ABB RobotStudio station: PROYECTO FINAL_TERMINADO_1.rsstn

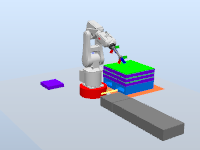
Station PROYECTO FINAL_TERMINADO (saved by RobotStudio 20.1.9014.1)
Controller Controller1, task T_ROB1: task frame (RAPID world) sits at (0, 0, 100) mm in the station
Controller Controller1
  mechanical unit ROB_1: IRB120_3_58__01, 6 joints, base frame (0, 0, 0) mm
Layout (positions relative to the parent item):
  - IRB120_3_58__01 [mechanism, from Robots\IRB120_3_58_G_01.rslib] at (0, 0, 100) mm; joint values [0, -0.0243, 0.3487, 0, 0.1992, 0] (rad or m)
  - soporte [mechanism, from biblioteca de robot\soporte.rslib] at (364.35, 0, 594) mm, rotated rx 180 ry 60 rz 180 deg
  - caja_modelo [part] at (-385.91, -352.84, 0) mm, rotated rx 0 ry 0 rz -0.36 deg
  - tapa_nueva3 [part] at (247.21, 259.23, 238) mm
  - pale_nuevo [part] at (30.71, 458.19, 106.32) mm
  - tapa_nueva2 [part] at (33.05, 460.18, 197.68) mm
  - tapa_nueva1 [part] at (31.05, 458.19, 150.3) mm
  - base_robot [part]
  - reposicion [smart component]
      signals: DI reseteo
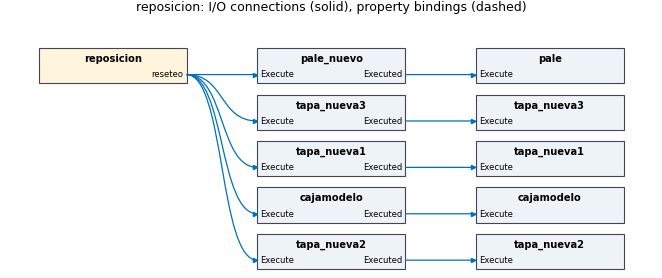
      connections:
        reposicion.reseteo -> pale_nuevo.Execute
        reposicion.reseteo -> tapa_nueva3.Execute
        reposicion.reseteo -> tapa_nueva1.Execute
        reposicion.reseteo -> cajamodelo.Execute
        reposicion.reseteo -> tapa_nueva2.Execute
        tapa_nueva2.Executed -> tapa_nueva2.Execute
        cajamodelo.Executed -> cajamodelo.Execute
        tapa_nueva1.Executed -> tapa_nueva1.Execute
        tapa_nueva3.Executed -> tapa_nueva3.Execute
        pale_nuevo.Executed -> pale.Execute
    - pale_nuevo [smart component, from Components\Positioner.rslib]
        properties: Object=pale_nuevo; Position=[0.061428 -0.45 0.13]; Orientation=[0 0 0]; Reference=Global; ReferenceObject=(none)
    - tapa_nueva1 [smart component, from Components\Positioner.rslib]
        properties: Object=tapa_nueva1; Position=[0.061428 -0.45 0.03]; Orientation=[0 0 0]; Reference=Global; ReferenceObject=(none)
    - tapa_nueva2 [smart component, from Components\Positioner.rslib]
        properties: Object=tapa_nueva2; Position=[0.061428 -0.45 0.018]; Orientation=[0 0 0]; Reference=Global; ReferenceObject=(none)
    - tapa_nueva3 [smart component, from Components\Positioner.rslib]
        properties: Object=tapa_nueva3; Position=[0.276428 -0.65 0]; Orientation=[0 0 0]; Reference=Global; ReferenceObject=(none)
    - cajamodelo [smart component, from Components\Positioner.rslib]
        properties: Object=(none); Position=[2.337542 0 0.14]; Orientation=[0 0 0]; Reference=Global; ReferenceObject=(none)
    - cajamodelo [smart component, from Components\Detacher.rslib]
        properties: Child=(none); KeepPosition=true
    - pale [smart component, from Components\Detacher.rslib]
        properties: Child=pale_nuevo; KeepPosition=true
    - tapa_nueva1 [smart component, from Components\Detacher.rslib]
        properties: Child=tapa_nueva1; KeepPosition=true
    - tapa_nueva2 [smart component, from Components\Detacher.rslib]
        properties: Child=tapa_nueva2; KeepPosition=true
    - tapa_nueva3 [smart component, from Components\Detacher.rslib]
        properties: Child=tapa_nueva3; KeepPosition=true
  - pedestal [part] at (28.42, 0, 0) mm
  - superficie [part] at (-277.21, 164.21, 2) mm
  - Pieza_3 [part]
  - tapa [part] at (246.05, 1411.93, 141.43) mm
  - cajas_y_banda [smart component]
      signals: DI caja_nuevaS, DO sensorLineal, DI attcherS, DI dettacherS, DI moverCajaS
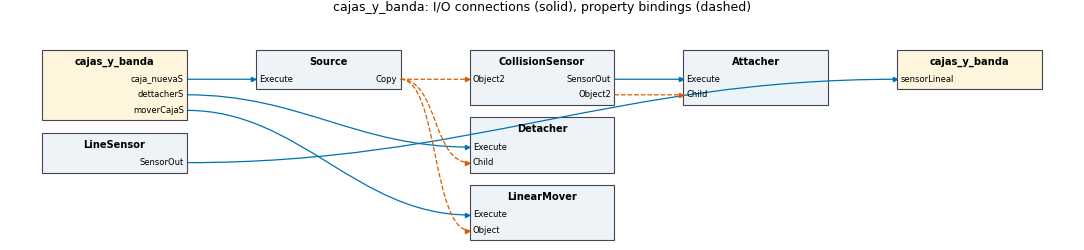
      connections:
        cajas_y_banda.caja_nuevaS -> Source.Execute
        LineSensor.SensorOut -> cajas_y_banda.sensorLineal
        cajas_y_banda.dettacherS -> Detacher.Execute
        cajas_y_banda.moverCajaS -> LinearMover.Execute
        CollisionSensor.SensorOut -> Attacher.Execute
        Source.Copy => Detacher.Child
        Source.Copy => CollisionSensor.Object2
        Source.Copy => LinearMover.Object
        CollisionSensor.Object2 => Attacher.Child
    - LineSensor [smart component, from Components\LineSensor.rslib] at (305.23, 54.67, 138.21) mm, rotated rx 90 ry 0 rz 0 deg
        properties: Start=[0.00491899596865375 -0.0182095563953858 -0.0453285878030492]; End=[0.00491899596865375 -0.0182095563953858 0.154671412196951]; Radius=0.005; SensedPart=(none); SensedPoint=[0 0 0]
      - _sensorPart_ [part]
    - LinearMover [smart component, from Components\LinearMover.rslib]
        properties: Object=caja_modelo_143; Direction=[-0.5 0 0]; Speed=0.3; Reference=Global; ReferenceObject=(none)
    - Source [smart component, from Components\Source.rslib]
        properties: Source=caja_modelo; Copy=caja_modelo_143; Parent=(none); Position=[1.18454 -0.1 0.1]; Orientation=[0 0 0]; Transient=false; PhysicsBehavior=0
    - CollisionSensor [smart component, from Components\CollisionSensor.rslib]
        properties: Object1=soporte; Object2=caja_modelo_143; NearMiss=0.002; Part1=(none); Part2=(none); CollisionType=0
    - Attacher [smart component, from Components\Attacher.rslib]
        properties: Parent=soporte; Flange=0; Child=caja_modelo_143; Mount=false; Offset=[0 0 0]; Orientation=[0 0 0]
    - Detacher [smart component, from Components\Detacher.rslib]
        properties: Child=caja_modelo_143; KeepPosition=true
  - pallet [smart component]
      connections:
        CollisionSensor.SensorOut -> Attacher.Execute
        CollisionSensor_2.SensorOut -> Detacher.Execute
    - Attacher [smart component, from Components\Attacher.rslib]
        properties: Parent=soporte; Flange=0; Child=pale_nuevo; Mount=false; Offset=[0 0 0]; Orientation=[0 0 0]
    - Detacher [smart component, from Components\Detacher.rslib]
        properties: Child=pale_nuevo; KeepPosition=true
    - CollisionSensor [smart component, from Components\CollisionSensor.rslib]
        properties: Object1=soporte; Object2=pale_nuevo; NearMiss=0.003; Part1=(none); Part2=(none); CollisionType=0
    - CollisionSensor_2 [smart component, from Components\CollisionSensor.rslib]
        properties: Object1=pale_nuevo; Object2=superficie; NearMiss=0.005; Part1=pale_nuevo; Part2=superficie; CollisionType=1
  - tapasDeNivel [smart component]
      signals: DI soltarTapa
      connections:
        CollisionSensor_3.SensorOut -> Attacher_2.Execute
        tapasDeNivel.soltarTapa -> Detacher_2.Execute
        CollisionSensor_4.SensorOut -> Attacher_3.Execute
        tapasDeNivel.soltarTapa -> Detacher_3.Execute
        CollisionSensor_5.SensorOut -> Attacher_4.Execute
        tapasDeNivel.soltarTapa -> Detacher_4.Execute
        CollisionSensor_3.Object2 => Attacher_2.Child
    - CollisionSensor_3 [smart component, from Components\CollisionSensor.rslib]
        properties: Object1=soporte; Object2=tapa_nueva1; NearMiss=0.001; Part1=(none); Part2=(none); CollisionType=0
    - Attacher_2 [smart component, from Components\Attacher.rslib]
        properties: Parent=soporte; Flange=0; Child=tapa_nueva1; Mount=false; Offset=[0 0 0]; Orientation=[0 0 0]
    - Detacher_2 [smart component, from Components\Detacher.rslib]
        properties: Child=tapa_nueva1; KeepPosition=true
    - Attacher_3 [smart component, from Components\Attacher.rslib]
        properties: Parent=soporte; Flange=0; Child=tapa_nueva2; Mount=false; Offset=[0 0 0]; Orientation=[0 0 0]
    - Detacher_3 [smart component, from Components\Detacher.rslib]
        properties: Child=tapa_nueva2; KeepPosition=true
    - CollisionSensor_4 [smart component, from Components\CollisionSensor.rslib]
        properties: Object1=soporte; Object2=tapa_nueva2; NearMiss=0.002; Part1=(none); Part2=(none); CollisionType=0
    - CollisionSensor_5 [smart component, from Components\CollisionSensor.rslib]
        properties: Object1=soporte; Object2=tapa_nueva3; NearMiss=0.001; Part1=(none); Part2=(none); CollisionType=0
    - Attacher_4 [smart component, from Components\Attacher.rslib]
        properties: Parent=soporte; Flange=0; Child=tapa_nueva3; Mount=false; Offset=[0 0 0]; Orientation=[0 0 0]
    - Detacher_4 [smart component, from Components\Detacher.rslib]
        properties: Child=tapa_nueva3; KeepPosition=true
  - Pieza_5 [part]
  - caja_modelo_132 [part] at (26.34, 258.19, 103.21) mm
  - caja_modelo_133 [part] at (27.58, 462.18, 103.22) mm
  - caja_modelo_134 [part] at (246.58, 460.85, 104.1) mm
  - caja_modelo_135 [part] at (245.34, 256.85, 104.3) mm
  - caja_modelo_136 [part] at (26.05, 460.19, 150.63) mm
  - caja_modelo_137 [part] at (245.05, 460.19, 150.37) mm
  - caja_modelo_138 [part] at (26.05, 256.19, 150.37) mm
  - caja_modelo_139 [part] at (245.05, 256.19, 150.61) mm
  - caja_modelo_140 [part] at (28.05, 462.19, 198.99) mm
  - caja_modelo_141 [part] at (248.85, 462.19, 199.65) mm
  - caja_modelo_142 [part] at (28.05, 258.19, 199.59) mm
  - caja_modelo_143 [part] at (247.05, 258.19, 199.43) mm
Attachment: soporte is attached to IRB120_3_58__01 / Link6
Station signals: DI inicioS, DI repo
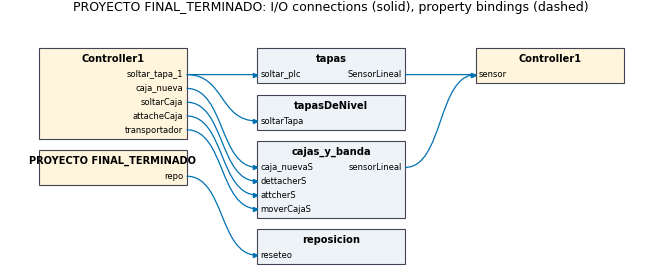
Station logic (signal -> signal, property => property):
  Controller1.soltar_tapa_1 -> tapas.soltar_plc
  anclado_y_desanclado_caja_modelo.SensorLineal -> Controller1.sensor
  cajas_y_banda.sensorLineal -> Controller1.sensor
  Controller1.caja_nueva -> cajas_y_banda.caja_nuevaS
  Controller1.soltarCaja -> cajas_y_banda.dettacherS
  Controller1.attacheCaja -> cajas_y_banda.attcherS
  Controller1.transportador -> cajas_y_banda.moverCajaS
  Controller1.soltar_tapa_1 -> tapasDeNivel.soltarTapa
  PROYECTO FINAL_TERMINADO.repo -> reposicion.reseteo
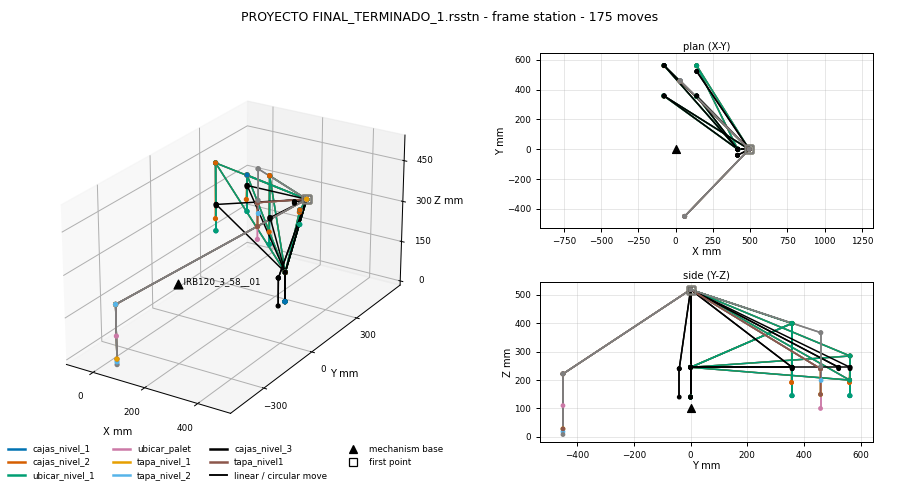
[picture p0: tool path of PROYECTO FINAL_TERMINADO_1.rsstn in frame station, 175 of 175 moves have a stored position in this frame; points joined in program order, loops and branches not executed]
Targets, tools, work objects and paths stored in the station, written as RAPID:
! task T_ROB1
MODULE CalibData
  PERS tooldata soporte:=[TRUE,[[0,0,150],[1,0,0,0]],[0.1,[0,0,1],[1,0,0,0],0,0,0]];
ENDMODULE

! task T_ROB1
MODULE Module1
  CONST robtarget pale_enposicion:=[[30.714,458.188,0],[0,1,0,0],[0,0,-2,0],[9E+09,9E+09,9E+09,9E+09,9E+09,9E+09]];
  CONST robtarget pale_enposicion_cercano:=[[30.714,458.188,140],[0,1,0,0],[0,0,-2,0],[9E+09,9E+09,9E+09,9E+09,9E+09,9E+09]];
  CONST robtarget home:=[[494.25763964,0,419],[0.5,0,0.866025404,0],[0,0,0,0],[9E+09,9E+09,9E+09,9E+09,9E+09,9E+09]];
  CONST robtarget tapa_nueva_3:=[[61.428,-450,-92],[0,1,0,0],[-1,0,1,0],[9E+09,9E+09,9E+09,9E+09,9E+09,9E+09]];
  CONST robtarget pale_nuevo:=[[61.428,-450,10],[0,1,0,0],[0,0,0,0],[9E+09,9E+09,9E+09,9E+09,9E+09,9E+09]];
  CONST robtarget tapa_nueva_1:=[[61.428,-450,-72],[0,1,0,0],[0,0,0,0],[9E+09,9E+09,9E+09,9E+09,9E+09,9E+09]];
  CONST robtarget tapa_nueva_2:=[[61.428,-450,-82],[0,1,0,0],[-1,0,1,0],[9E+09,9E+09,9E+09,9E+09,9E+09,9E+09]];
  CONST robtarget home_1:=[[417.312,0.001,268.837186077],[0,1,0,0],[0,0,-2,0],[9E+09,9E+09,9E+09,9E+09,9E+09,9E+09]];
  CONST robtarget cercano_pale_nuevo:=[[61.428,-450,121.709],[0,1,0,0],[-1,0,1,0],[9E+09,9E+09,9E+09,9E+09,9E+09,9E+09]];
  CONST robtarget tapa_1_en_posicion:=[[31.052,458.187,49.432],[0,1,0,0],[0,0,-2,0],[9E+09,9E+09,9E+09,9E+09,9E+09,9E+09]];
  CONST robtarget tomar_caja_de_banda:=[[417.64,0,40],[0,1,0,0],[0,0,-2,0],[9E+09,9E+09,9E+09,9E+09,9E+09,9E+09]];
  CONST robtarget punto_cercano_banda:=[[417.652,0,145],[0,1,0,0],[0,0,-2,0],[9E+09,9E+09,9E+09,9E+09,9E+09,9E+09]];
  CONST robtarget lugar4_primerNivel:=[[140.837,356.854,44.894],[0,1,0,0],[0,0,-2,0],[9E+09,9E+09,9E+09,9E+09,9E+09,9E+09]];
  CONST robtarget lugar3_primerNivel:=[[142.08,560.85,44.894],[0,1,0,0],[0,0,-2,0],[9E+09,9E+09,9E+09,9E+09,9E+09,9E+09]];
  CONST robtarget lugar2_primerNivel:=[[-76.917,562.181,44.879],[0,1,0,0],[1,0,-1,0],[9E+09,9E+09,9E+09,9E+09,9E+09,9E+09]];
  CONST robtarget lugar1_primerNivel:=[[-78.159,358.191,44.894],[0,1,0,0],[1,0,-1,0],[9E+09,9E+09,9E+09,9E+09,9E+09,9E+09]];
  CONST robtarget cuadrante1:=[[-78.159,358.191,300],[0,1,0,0],[1,0,-1,0],[9E+09,9E+09,9E+09,9E+09,9E+09,9E+09]];
  CONST robtarget cuadrante2:=[[-76.917,562.181,185],[0,1,0,0],[1,0,-1,0],[9E+09,9E+09,9E+09,9E+09,9E+09,9E+09]];
  CONST robtarget cuadrante3:=[[142.08,560.85,100],[0,1,0,0],[0,0,-2,0],[9E+09,9E+09,9E+09,9E+09,9E+09,9E+09]];
  CONST robtarget cuadrante4:=[[140.837,356.854,300],[0,1,0,0],[0,0,-2,0],[9E+09,9E+09,9E+09,9E+09,9E+09,9E+09]];
  CONST robtarget lugar3_segundoNivel:=[[-78.448,356.187,91.479],[0,1,0,0],[1,0,-1,0],[9E+09,9E+09,9E+09,9E+09,9E+09,9E+09]];
  CONST robtarget lugar1_segundoNivel:=[[-78.448,560.187,91.479],[0,1,0,0],[1,0,-1,0],[9E+09,9E+09,9E+09,9E+09,9E+09,9E+09]];
  CONST robtarget lugar2_segundoNivel:=[[140.552,560.187,91.479],[0,1,0,0],[0,0,-2,0],[9E+09,9E+09,9E+09,9E+09,9E+09,9E+09]];
  CONST robtarget lugar4_segundoNivel:=[[140.552,356.187,91.479],[0,1,0,0],[0,0,-2,0],[9E+09,9E+09,9E+09,9E+09,9E+09,9E+09]];
  CONST robtarget home_2:=[[494.25763964,0,419],[0.5,0,0.866025404,0],[0,0,0,0],[9E+09,9E+09,9E+09,9E+09,9E+09,9E+09]];
  CONST robtarget home_3:=[[494.25763964,0,419],[0.5,0,0.866025404,0],[0,0,0,0],[9E+09,9E+09,9E+09,9E+09,9E+09,9E+09]];
  CONST robtarget punto_cercano_banda_2:=[[417.652,0,145],[0,1,0,0],[0,0,-2,0],[9E+09,9E+09,9E+09,9E+09,9E+09,9E+09]];
  CONST robtarget tomar_caja_de_banda_2:=[[417.652,0,45],[0,1,0,0],[0,0,-2,0],[9E+09,9E+09,9E+09,9E+09,9E+09,9E+09]];
  CONST robtarget cuadrante2_2:=[[-76.917,562.181,185],[0,1,0,0],[1,0,-1,0],[9E+09,9E+09,9E+09,9E+09,9E+09,9E+09]];
  CONST robtarget lugar1_segundoNivel_2:=[[-78.448,560.187,91.479],[0,1,0,0],[1,0,-1,0],[9E+09,9E+09,9E+09,9E+09,9E+09,9E+09]];
  CONST robtarget cuadrante3_2:=[[142.08,560.85,100],[0,1,0,0],[0,0,-2,0],[9E+09,9E+09,9E+09,9E+09,9E+09,9E+09]];
  CONST robtarget lugar2_segundoNivel_2:=[[140.552,560.187,91.479],[0,1,0,0],[0,0,-2,0],[9E+09,9E+09,9E+09,9E+09,9E+09,9E+09]];
  CONST robtarget home_2_2:=[[494.25763964,0,419],[0.5,0,0.866025404,0],[0,0,0,0],[9E+09,9E+09,9E+09,9E+09,9E+09,9E+09]];
  CONST robtarget tapa_nueva_enPosicion:=[[33.052,460.186,98.754],[0,1,0,0],[0,0,-2,0],[9E+09,9E+09,9E+09,9E+09,9E+09,9E+09]];
  CONST robtarget lugar3_tercerNivel:=[[-76.448,358.186,140.032],[0,1,0,0],[0,0,0,0],[9E+09,9E+09,9E+09,9E+09,9E+09,9E+09]];
  CONST robtarget lugar4_tercernivel:=[[142.552,358.186,140.032],[0,1,0,0],[0,0,-2,0],[9E+09,9E+09,9E+09,9E+09,9E+09,9E+09]];
  CONST robtarget lugar2_tercerNivel:=[[142.552,522.186,140.032],[0,1,0,0],[0,0,-2,0],[9E+09,9E+09,9E+09,9E+09,9E+09,9E+09]];
  CONST robtarget lugar1_tercerNivel:=[[-76.448,562.186,140.032],[0,1,0,0],[0,0,0,0],[9E+09,9E+09,9E+09,9E+09,9E+09,9E+09]];
  CONST robtarget cuadrante2_tercerNivel:=[[142.552,522.186,145],[0,1,0,0],[0,0,0,0],[9E+09,9E+09,9E+09,9E+09,9E+09,9E+09]];
  CONST robtarget cuadrante1_tercerNivel:=[[-76.448,562.186,145],[0,1,0,0],[0,0,0,0],[9E+09,9E+09,9E+09,9E+09,9E+09,9E+09]];
  CONST robtarget cuadrante3_tercerNivel:=[[-76.448,358.186,145],[0,1,0,0],[0,0,0,0],[9E+09,9E+09,9E+09,9E+09,9E+09,9E+09]];
  CONST robtarget cuadrante4_tercerNivel:=[[142.552,358.186,145],[0,1,0,0],[0,0,0,0],[9E+09,9E+09,9E+09,9E+09,9E+09,9E+09]];
  CONST robtarget punto_cercano_banda_3:=[[494.25763964,0,519],[0.5,0,0.866025404,0],[0,0,0,0],[9E+09,9E+09,9E+09,9E+09,9E+09,9E+09]];
  CONST robtarget tomar_cajaEsquina:=[[415.84,-40,40],[0,1,0,0],[-1,0,1,0],[9E+09,9E+09,9E+09,9E+09,9E+09,9E+09]];
  CONST robtarget cerca_cajaEsquina:=[[415.84,-40,140],[0,1,0,0],[-1,0,1,0],[9E+09,9E+09,9E+09,9E+09,9E+09,9E+09]];
  CONST robtarget fijar_tapa3:=[[51.851,458.186,148.595],[0,1,0,0],[0,0,-2,0],[9E+09,9E+09,9E+09,9E+09,9E+09,9E+09]];
  CONST robtarget aprox_fijarTapa3:=[[51.851,458.186,173.199585424],[0,1,0,0],[0,0,-2,0],[9E+09,9E+09,9E+09,9E+09,9E+09,9E+09]];
  CONST robtarget Target_10:=[[32.215,459.23,148.852],[0,1,0,0],[0,0,-2,0],[9E+09,9E+09,9E+09,9E+09,9E+09,9E+09]];
  CONST robtarget Target_20:=[[32.215,459.23,267.1643111],[0,1,0,0],[0,0,-2,0],[9E+09,9E+09,9E+09,9E+09,9E+09,9E+09]];
  PROC cajas_nivel_1()
    WaitDI paso,1;
    MoveL home,v300,fine,soporte\WObj:=wobj0;
    MoveL punto_cercano_banda,v300,fine,soporte\WObj:=wobj0;
    MoveL tomar_caja_de_banda,v300,fine,soporte\WObj:=wobj0;
    MoveL punto_cercano_banda,v300,fine,soporte\WObj:=wobj0;
    MoveL cuadrante1,v300,fine,soporte\WObj:=wobj0;
    MoveL lugar1_primerNivel,v300,fine,soporte\WObj:=wobj0;
    MoveL cuadrante1,v300,fine,soporte\WObj:=wobj0;
    MoveL home,v300,fine,soporte\WObj:=wobj0;
    WaitDI paso,1;
    MoveL home,v300,fine,soporte\WObj:=wobj0;
    MoveL punto_cercano_banda,v300,fine,soporte\WObj:=wobj0;
    MoveL tomar_caja_de_banda,v300,fine,soporte\WObj:=wobj0;
    MoveL punto_cercano_banda,v300,fine,soporte\WObj:=wobj0;
    MoveL cuadrante2,v300,fine,soporte\WObj:=wobj0;
    MoveL lugar2_primerNivel,v300,fine,soporte\WObj:=wobj0;
    MoveL cuadrante2,v300,fine,soporte\WObj:=wobj0;
    MoveL home,v300,fine,soporte\WObj:=wobj0;
    WaitDI paso,1;
    MoveL home,v300,fine,soporte\WObj:=wobj0;
    MoveL punto_cercano_banda,v300,fine,soporte\WObj:=wobj0;
    MoveL tomar_caja_de_banda,v300,fine,soporte\WObj:=wobj0;
    MoveL punto_cercano_banda,v300,fine,soporte\WObj:=wobj0;
    MoveL cuadrante3,v300,fine,soporte\WObj:=wobj0;
    MoveL lugar3_primerNivel,v300,fine,soporte\WObj:=wobj0;
    MoveL cuadrante3,v300,fine,soporte\WObj:=wobj0;
    MoveL home,v300,fine,soporte\WObj:=wobj0;
    WaitDI paso,1;
    MoveL home,v300,fine,soporte\WObj:=wobj0;
    MoveL punto_cercano_banda,v300,fine,soporte\WObj:=wobj0;
    MoveL tomar_caja_de_banda,v300,fine,soporte\WObj:=wobj0;
    MoveL punto_cercano_banda,v300,fine,soporte\WObj:=wobj0;
    MoveL cuadrante4,v300,fine,soporte\WObj:=wobj0;
    MoveL lugar4_primerNivel,v300,fine,soporte\WObj:=wobj0;
    MoveL cuadrante4,v300,fine,soporte\WObj:=wobj0;
    MoveL home,v300,fine,soporte\WObj:=wobj0;
  ENDPROC
  PROC main()
    WaitDI inicio,1;
    ubicar_palet;
    ubicar_nivel_1;
    tapa_nivel_1;
    cajas_nivel_2;
    tapa_nivel_2;
    cajas_nivel_3;
    tapar_nivel3;
  ENDPROC
  PROC cajas_nivel_2()
    SetDO caja_nueva,1;
    SetDO caja_nueva,0;
    SetDO transportador,1;
    WaitDI sensor,1;
    SetDO transportador,0;
    WaitDI sensor,1;
    MoveL home,v300,fine,soporte\WObj:=wobj0;
    MoveL punto_cercano_banda,v300,fine,soporte\WObj:=wobj0;
    WaitDI sensor,1;
    MoveL tomar_caja_de_banda,v300,fine,soporte\WObj:=wobj0;
    MoveL punto_cercano_banda,v300,fine,soporte\WObj:=wobj0;
    MoveL cuadrante2,v300,fine,soporte\WObj:=wobj0;
    MoveL lugar1_segundoNivel,v300,fine,soporte\WObj:=wobj0;
    SetDO soltarCaja,1;
    SetDO soltarCaja,0;
    MoveL cuadrante2,v300,fine,soporte\WObj:=wobj0;
    MoveL home,v300,fine,soporte\WObj:=wobj0;
    SetDO caja_nueva,1;
    SetDO caja_nueva,0;
    SetDO transportador,1;
    WaitDI sensor,1;
    SetDO transportador,0;
    WaitDI sensor,1;
    MoveL home,v300,fine,soporte\WObj:=wobj0;
    MoveL punto_cercano_banda,v300,fine,soporte\WObj:=wobj0;
    WaitDI sensor,1;
    MoveL tomar_caja_de_banda,v300,fine,soporte\WObj:=wobj0;
    MoveL punto_cercano_banda,v300,fine,soporte\WObj:=wobj0;
    MoveL cuadrante3,v300,fine,soporte\WObj:=wobj0;
    MoveL lugar2_segundoNivel,v300,fine,soporte\WObj:=wobj0;
    SetDO soltarCaja,1;
    SetDO soltarCaja,0;
    MoveL cuadrante3,v300,fine,soporte\WObj:=wobj0;
    MoveL home,v300,fine,soporte\WObj:=wobj0;
    SetDO caja_nueva,1;
    SetDO caja_nueva,0;
    SetDO transportador,1;
    WaitDI sensor,1;
    SetDO transportador,0;
    WaitDI sensor,1;
    MoveL home,v300,fine,soporte\WObj:=wobj0;
    MoveL punto_cercano_banda_2,v300,fine,soporte\WObj:=wobj0;
    WaitDI sensor,1;
    MoveL tomar_caja_de_banda,v300,fine,soporte\WObj:=wobj0;
    MoveL punto_cercano_banda,v300,fine,soporte\WObj:=wobj0;
    MoveL cuadrante1,v300,fine,soporte\WObj:=wobj0;
    MoveL lugar3_segundoNivel,v300,fine,soporte\WObj:=wobj0;
    SetDO soltarCaja,1;
    SetDO soltarCaja,0;
    MoveL cuadrante1,v300,fine,soporte\WObj:=wobj0;
    MoveL home,v300,fine,soporte\WObj:=wobj0;
    SetDO caja_nueva,1;
    SetDO caja_nueva,0;
    SetDO transportador,1;
    WaitDI sensor,1;
    SetDO transportador,0;
    WaitDI sensor,1;
    MoveL home,v300,fine,soporte\WObj:=wobj0;
    MoveL punto_cercano_banda,v300,fine,soporte\WObj:=wobj0;
    MoveL tomar_caja_de_banda,v300,fine,soporte\WObj:=wobj0;
    MoveL punto_cercano_banda,v300,fine,soporte\WObj:=wobj0;
    MoveL cuadrante4,v300,fine,soporte\WObj:=wobj0;
    MoveL lugar4_segundoNivel,v300,fine,soporte\WObj:=wobj0;
    SetDO soltarCaja,1;
    SetDO soltarCaja,0;
    MoveL cuadrante4,v300,fine,soporte\WObj:=wobj0;
    MoveL home,v300,fine,soporte\WObj:=wobj0;
  ENDPROC
  PROC ubicar_nivel_1()
    SetDO caja_nueva,1;
    SetDO caja_nueva,0;
    SetDO transportador,1;
    WaitDI sensor,1;
    SetDO transportador,0;
    WaitDI sensor,1;
    MoveL home,v500,fine,soporte\WObj:=wobj0;
    MoveL punto_cercano_banda,v500,fine,soporte\WObj:=wobj0;
    WaitDI sensor,1;
    MoveL tomar_caja_de_banda,v500,fine,soporte\WObj:=wobj0;
    MoveL punto_cercano_banda,v500,fine,soporte\WObj:=wobj0;
    MoveL cuadrante1,v500,fine,soporte\WObj:=wobj0;
    MoveL lugar1_primerNivel,v500,fine,soporte\WObj:=wobj0;
    SetDO soltarCaja,1;
    SetDO soltarCaja,0;
    MoveL cuadrante1,v500,fine,soporte\WObj:=wobj0;
    MoveL home,v500,fine,soporte\WObj:=wobj0;
    SetDO caja_nueva,1;
    SetDO caja_nueva,0;
    SetDO transportador,1;
    WaitDI sensor,1;
    SetDO transportador,0;
    MoveL home,v500,fine,soporte\WObj:=wobj0;
    MoveL punto_cercano_banda,v500,fine,soporte\WObj:=wobj0;
    WaitDI sensor,1;
    MoveL tomar_caja_de_banda,v500,fine,soporte\WObj:=wobj0;
    MoveL punto_cercano_banda,v500,fine,soporte\WObj:=wobj0;
    MoveL cuadrante2,v500,fine,soporte\WObj:=wobj0;
    MoveL lugar2_primerNivel,v500,fine,soporte\WObj:=wobj0;
    SetDO soltarCaja,1;
    SetDO soltarCaja,0;
    MoveL cuadrante2,v500,fine,soporte\WObj:=wobj0;
    MoveL home,v500,fine,soporte\WObj:=wobj0;
    SetDO caja_nueva,1;
    SetDO caja_nueva,0;
    SetDO transportador,1;
    WaitDI sensor,1;
    SetDO transportador,0;
    MoveL home,v500,fine,soporte\WObj:=wobj0;
    MoveL punto_cercano_banda,v500,fine,soporte\WObj:=wobj0;
    WaitDI sensor,1;
    MoveL tomar_caja_de_banda,v500,fine,soporte\WObj:=wobj0;
    MoveL punto_cercano_banda,v500,fine,soporte\WObj:=wobj0;
    MoveL cuadrante3,v500,fine,soporte\WObj:=wobj0;
    MoveL lugar3_primerNivel,v500,fine,soporte\WObj:=wobj0;
    SetDO soltarCaja,1;
    SetDO soltarCaja,0;
    MoveL cuadrante3,v500,fine,soporte\WObj:=wobj0;
    MoveL home,v500,fine,soporte\WObj:=wobj0;
    SetDO caja_nueva,1;
    SetDO caja_nueva,0;
    SetDO transportador,1;
    WaitDI sensor,1;
    SetDO transportador,0;
    MoveL home,v500,fine,soporte\WObj:=wobj0;
    MoveL punto_cercano_banda,v500,fine,soporte\WObj:=wobj0;
    WaitDI sensor,1;
    MoveL tomar_caja_de_banda,v500,fine,soporte\WObj:=wobj0;
    MoveL punto_cercano_banda,v500,fine,soporte\WObj:=wobj0;
    MoveL cuadrante4,v500,fine,soporte\WObj:=wobj0;
    MoveL lugar4_primerNivel,v500,fine,soporte\WObj:=wobj0;
    SetDO soltarCaja,1;
    SetDO soltarCaja,0;
    MoveL cuadrante4,v500,fine,soporte\WObj:=wobj0;
    MoveL home,v500,fine,soporte\WObj:=wobj0;
  ENDPROC
  PROC Path_10()
    tapa_nivel_2;
  ENDPROC
  PROC ubicar_palet()
    MoveL home,v300,fine,soporte\WObj:=wobj0;
    MoveL cercano_pale_nuevo,v300,fine,soporte\WObj:=wobj0;
    MoveL pale_nuevo,v300,fine,soporte\WObj:=wobj0;
    MoveL cercano_pale_nuevo,v300,fine,soporte\WObj:=wobj0;
    MoveL home,v300,fine,soporte\WObj:=wobj0;
    MoveL pale_enposicion_cercano,v300,fine,soporte\WObj:=wobj0;
    MoveL pale_enposicion,v300,fine,soporte\WObj:=wobj0;
    MoveL pale_enposicion_cercano,v300,fine,soporte\WObj:=wobj0;
    MoveL home,v300,fine,soporte\WObj:=wobj0;
  ENDPROC
  PROC tapa_nivel_1()
    MoveL home,v500,fine,soporte\WObj:=wobj0;
    MoveL cercano_pale_nuevo,v500,fine,soporte\WObj:=wobj0;
    MoveL tapa_nueva_1,v500,fine,soporte\WObj:=wobj0;
    MoveL cercano_pale_nuevo,v500,fine,soporte\WObj:=wobj0;
    MoveL home,v500,fine,soporte\WObj:=wobj0;
    MoveL pale_enposicion_cercano,v500,fine,soporte\WObj:=wobj0;
    MoveL tapa_1_en_posicion,v500,fine,soporte\WObj:=wobj0;
    SetDO soltar_tapa_1,1;
    SetDO soltar_tapa_1,0;
    MoveL pale_enposicion_cercano,v500,fine,soporte\WObj:=wobj0;
    MoveL home,v500,fine,soporte\WObj:=wobj0;
  ENDPROC
  PROC tapa_nivel_2()
    MoveL home,v500,fine,soporte\WObj:=wobj0;
    MoveL cercano_pale_nuevo,v500,fine,soporte\WObj:=wobj0;
    MoveL tapa_nueva_2,v500,fine,soporte\WObj:=wobj0;
    MoveL cercano_pale_nuevo,v500,fine,soporte\WObj:=wobj0;
    MoveL home,v500,fine,soporte\WObj:=wobj0;
    MoveL pale_enposicion_cercano,v500,fine,soporte\WObj:=wobj0;
    MoveL tapa_nueva_enPosicion,v500,fine,soporte\WObj:=wobj0;
    SetDO soltar_tapa_1,1;
    SetDO soltar_tapa_1,0;
    MoveL pale_enposicion_cercano,v500,fine,soporte\WObj:=wobj0;
    MoveL home,v500,fine,soporte\WObj:=wobj0;
  ENDPROC
  PROC cajas_nivel_3()
    SetDO caja_nueva,1;
    SetDO caja_nueva,0;
    SetDO transportador,1;
    WaitDI sensor,1;
    SetDO transportador,0;
    WaitDI sensor,1;
    MoveL home,v500,fine,soporte\WObj:=wobj0;
    MoveL punto_cercano_banda,v500,fine,soporte\WObj:=wobj0;
    WaitDI sensor,1;
    MoveL tomar_caja_de_banda,v500,fine,soporte\WObj:=wobj0;
    MoveL punto_cercano_banda,v500,fine,soporte\WObj:=wobj0;
    MoveL cuadrante1_tercerNivel,v500,fine,soporte\WObj:=wobj0;
    MoveL lugar1_tercerNivel,v500,fine,soporte\WObj:=wobj0;
    SetDO soltarCaja,1;
    SetDO soltarCaja,0;
    MoveL cuadrante1_tercerNivel,v500,fine,soporte\WObj:=wobj0;
    MoveL home,v500,fine,soporte\WObj:=wobj0;
    SetDO caja_nueva,1;
    SetDO caja_nueva,0;
    SetDO transportador,1;
    WaitDI sensor,1;
    SetDO transportador,0;
    WaitDI sensor,1;
    MoveL home,v500,fine,soporte\WObj:=wobj0;
    MoveL cerca_cajaEsquina,v500,fine,soporte\WObj:=wobj0;
    WaitDI sensor,1;
    MoveL cerca_cajaEsquina,v500,fine,soporte\WObj:=wobj0;
    MoveL tomar_cajaEsquina,v500,fine,soporte\WObj:=wobj0;
    MoveL cerca_cajaEsquina,v500,fine,soporte\WObj:=wobj0;
    MoveL home,v500,fine,soporte\WObj:=wobj0;
    MoveL cuadrante2_tercerNivel,v500,fine,soporte\WObj:=wobj0;
    MoveL lugar2_tercerNivel,v500,fine,soporte\WObj:=wobj0;
    SetDO soltarCaja,1;
    SetDO soltarCaja,0;
    MoveL cuadrante2_tercerNivel,v500,fine,soporte\WObj:=wobj0;
    MoveL home,v500,fine,soporte\WObj:=wobj0;
    SetDO caja_nueva,1;
    SetDO caja_nueva,0;
    SetDO transportador,1;
    WaitDI sensor,1;
    SetDO transportador,0;
    WaitDI sensor,1;
    MoveL home,v500,fine,soporte\WObj:=wobj0;
    MoveL punto_cercano_banda,v500,fine,soporte\WObj:=wobj0;
    WaitDI sensor,1;
    MoveL tomar_caja_de_banda,v500,fine,soporte\WObj:=wobj0;
    MoveL punto_cercano_banda,v500,fine,soporte\WObj:=wobj0;
    MoveL cuadrante3_tercerNivel,v500,fine,soporte\WObj:=wobj0;
    MoveL lugar3_tercerNivel,v500,fine,soporte\WObj:=wobj0;
    SetDO soltarCaja,1;
    SetDO soltarCaja,0;
    MoveL cuadrante3_tercerNivel,v500,fine,soporte\WObj:=wobj0;
    MoveL home,v500,fine,soporte\WObj:=wobj0;
    SetDO caja_nueva,1;
    SetDO caja_nueva,0;
    SetDO transportador,1;
    WaitDI sensor,1;
    SetDO transportador,0;
    WaitDI sensor,1;
    MoveL home,v500,fine,soporte\WObj:=wobj0;
    MoveL punto_cercano_banda,v500,fine,soporte\WObj:=wobj0;
    WaitDI sensor,1;
    MoveL tomar_caja_de_banda,v500,fine,soporte\WObj:=wobj0;
    MoveL punto_cercano_banda,v500,fine,soporte\WObj:=wobj0;
    MoveL cuadrante4_tercerNivel,v500,fine,soporte\WObj:=wobj0;
    MoveL lugar4_tercernivel,v500,fine,soporte\WObj:=wobj0;
    SetDO soltarCaja,1;
    SetDO soltarCaja,0;
    MoveL cuadrante4_tercerNivel,v500,fine,soporte\WObj:=wobj0;
    MoveL home,v500,fine,soporte\WObj:=wobj0;
  ENDPROC
  PROC tapa_nivel1()
    MoveL home,v1000,z100,soporte\WObj:=wobj0;
    MoveL cercano_pale_nuevo,v1000,z100,soporte\WObj:=wobj0;
    MoveL tapa_nueva_1,v1000,z100,soporte\WObj:=wobj0;
    MoveL cercano_pale_nuevo,v1000,z100,soporte\WObj:=wobj0;
    MoveL home,v1000,z100,soporte\WObj:=wobj0;
    MoveL pale_enposicion_cercano,v1000,z100,soporte\WObj:=wobj0;
    MoveL tapa_1_en_posicion,v1000,z100,soporte\WObj:=wobj0;
    MoveL pale_enposicion_cercano,v1000,z100,soporte\WObj:=wobj0;
    MoveL home,v1000,z100,soporte\WObj:=wobj0;
  ENDPROC
  PROC tapar_nivel3()
    MoveL home,v500,fine,soporte\WObj:=wobj0;
    MoveL cercano_pale_nuevo,v500,fine,soporte\WObj:=wobj0;
    MoveL tapa_nueva_3,v500,fine,soporte\WObj:=wobj0;
    MoveL cercano_pale_nuevo,v500,fine,soporte\WObj:=wobj0;
    MoveL home,v500,fine,soporte\WObj:=wobj0;
    MoveL Target_20,v1000,fine,soporte\WObj:=wobj0;
    MoveL Target_10,v1000,fine,soporte\WObj:=wobj0;
    SetDO soltar_tapa_1,1;
    SetDO soltar_tapa_1,0;
    MoveL Target_20,v1000,fine,soporte\WObj:=wobj0;
    MoveL home,v500,fine,soporte\WObj:=wobj0;
  ENDPROC
ENDMODULE

